// TIA Portal V20 export
DATA_BLOCK "BK17"   // DB263
// stored: MemoryReserve 100
   VAR
      "X10-1 LASER MARKING COVER UP" : Bool;
      "X10-2 LASER MARKING COVER DOWN" : Bool;
      "X12-1 LASER MARKING Stage Lift UP" : Bool;
      "X12-2 LASER MARKING Stage Lift DOWN" : Bool;
      "X14-1 SPARE" : Bool;
      "X14-2 LASER MARKING STACK DETECT SENSOR" : Bool;
      "X16-1 SPARE" : Bool;
      "X16-2 SPARE" : Bool;
   END_VAR
BEGIN
END_DATA_BLOCK
